// TIA Portal V20 export
FUNCTION_BLOCK "FB_Start_Test"   // FB5, LAD
{ S7_Optimized_Access := 'TRUE' }
// stored: MemoryReserve 100, SetENOAutomatically false
   VAR_INPUT
      Button_Start_Approve : Bool;
      Electrical_Current_Test_Approved : Bool;
      Visual_Test_Approved_PLC : Bool;
      Reset_Funcional_Test : Bool;
   END_VAR
   VAR_OUTPUT
      Start_Functional_Test : Bool;
      Blink_Button_Light : Bool;
      Turn_On_Button_Light : Bool;
      Light_Fail_Test : Bool;
      Light_Approve_Test : Bool;
   END_VAR
   VAR
      Aux_Trigger_0 : Bool;
   END_VAR
   VAR_TEMP   // added for the SCL form of the ladder/FBD networks
      _w1 : Bool;
      _w2 : Bool;
   END_VAR
BEGIN

REGION Network 1: Set Start Functional Test, Blink the Button Light, Turn on Red Light (Fail Test)
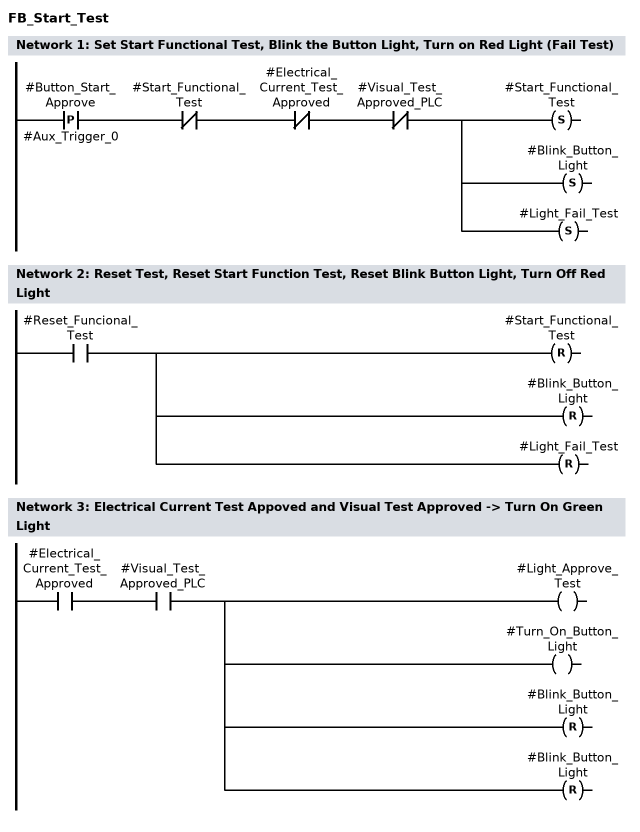
   RUNG wire#powerrail
      P_Contact(operand := #Button_Start_Approve, bit := #Aux_Trigger_0)
      I_Contact( #Start_Functional_Test )
      I_Contact( #Electrical_Current_Test_Approved )
      I_Contact( #Visual_Test_Approved_PLC )
      wire#w1
      S_Coil( #Start_Functional_Test )
   END_RUNG
   RUNG wire#w1
      S_Coil( #Blink_Button_Light )
   END_RUNG
   RUNG wire#w1
      S_Coil( #Light_Fail_Test )
   END_RUNG
   // the same network as SCL:
   #_w1 := #Button_Start_Approve AND NOT #Aux_Trigger_0;   // rising edge of #Button_Start_Approve
   #Aux_Trigger_0 := #Button_Start_Approve;
   #_w2 := #_w1 AND NOT #Start_Functional_Test AND NOT #Electrical_Current_Test_Approved AND NOT #Visual_Test_Approved_PLC;
   IF #_w2 THEN
       #Start_Functional_Test := TRUE;
       #Blink_Button_Light := TRUE;
       #Light_Fail_Test := TRUE;
   END_IF;
END_REGION

REGION Network 2: Reset Test, Reset Start Function Test, Reset Blink Button Light, Turn Off Red Light
   RUNG wire#powerrail
      Contact( #Reset_Funcional_Test )
      wire#w1
      R_Coil( #Start_Functional_Test )
   END_RUNG
   RUNG wire#w1
      R_Coil( #Blink_Button_Light )
   END_RUNG
   RUNG wire#w1
      R_Coil( #Light_Fail_Test )
   END_RUNG
   // the same network as SCL:
   IF #Reset_Funcional_Test THEN
       #Start_Functional_Test := FALSE;
       #Blink_Button_Light := FALSE;
       #Light_Fail_Test := FALSE;
   END_IF;
END_REGION

REGION Network 3: Electrical Current Test Appoved and Visual Test Approved -> Turn On Green Light
   RUNG wire#powerrail
      Contact( #Electrical_Current_Test_Approved )
      Contact( #Visual_Test_Approved_PLC )
      wire#w1
      Coil( #Light_Approve_Test )
   END_RUNG
   RUNG wire#w1
      Coil( #Turn_On_Button_Light )
   END_RUNG
   RUNG wire#w1
      R_Coil( #Blink_Button_Light )
   END_RUNG
   RUNG wire#w1
      R_Coil( #Blink_Button_Light )
   END_RUNG
   // the same network as SCL:
   #Light_Approve_Test := #Electrical_Current_Test_Approved AND #Visual_Test_Approved_PLC;
   #Turn_On_Button_Light := #Light_Approve_Test;
   IF #Light_Approve_Test THEN
       #Blink_Button_Light := FALSE;
       #Blink_Button_Light := FALSE;
   END_IF;
END_REGION
END_FUNCTION_BLOCK
